FUNCTION_BLOCK F_NOT
  {SET_ATTRIBUTE(OpcUa, Service)}
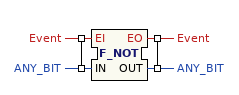
  EVENT_INPUT
    EI WITH IN;
  END_EVENT
  EVENT_OUTPUT
    EO WITH OUT;
  END_EVENT
  VAR_INPUT
    IN : ANY_BIT;
  END_VAR
  VAR_OUTPUT
    OUT : ANY_BIT;
  END_VAR
END_FUNCTION_BLOCK
